Staubli VAL3: onSave.pgx

public program onSave(string& x_sItem[])
begin
  // other option before save
end
